(* IEC 61131-3 sources: plc-browser-io/CODESYSv3/CODESYS_Control_Win_V3_x64/Application/Events, 1 file *)

(* ---- StartDone.st ---- *)
FUNCTION StartDone : DWORD
VAR_IN_OUT
	EventPrm: CmpApp.EVTPARAM_CmpApp;
END_VAR
VAR
END_VAR

// === IMPLEMENTATION ===
// Init logger component
LogComponent.Logger();

// Initialization Started
LogComponent.Logger.LogADD(Component:= LogComponent.RTM , LogClass:= cmplog.LogClass.LOG_INFO, Message:= 'Initialization started ');

// Initialization Ended
LogComponent.Logger.LogADD(Component:= LogComponent.RTM , LogClass:= cmplog.LogClass.LOG_INFO, Message:= 'Initialization ended');
